{attribute 'GeneratedUsingTerminal: EM7004-0000-9995'}
{attribute addProperty BoxType "EM7004-0000-9995"}
{attribute addProperty Id "CtrlAT %Q*UINT2ValueAT %Q*UINT2"}
{attribute addProperty CRC "3080298004"}
{attribute addProperty Size "4"}
TYPE Encoder_Channel_B7999E14 :
STRUCT
	{attribute addProperty Name "Ctrl"}
	Ctrl AT %Q* : UINT;
	{attribute addProperty Name "Value"}
	Value AT %Q* : UINT;
END_STRUCT
END_TYPE

(* stored: Version 1.2.0.0, ProductVersion 3.1.4024.9
   DUT Encoder_Channel_B7999E14: Id {de133ac4-5750-4b78-bd60-adb7c0d56fe4} *)
